FUNCTION_BLOCK E_F_TRIG
  (* Version 1.0, 2005-07-05, Goran Cengic, Chalmers *)
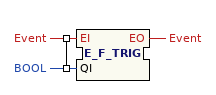
  EVENT_INPUT
    EI WITH QI;
  END_EVENT
  EVENT_OUTPUT
    EO;
  END_EVENT
  VAR_INPUT
    QI : BOOL;
  END_VAR
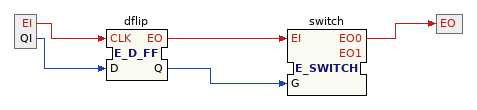
  FBS
    dflip : E_D_FF;
    switch : E_SWITCH;
  END_FBS
  EVENT_CONNECTIONS
    EI TO dflip.CLK;
    dflip.EO TO switch.EI;
    switch.EO0 TO EO;
  END_CONNECTIONS
  DATA_CONNECTIONS
    QI TO dflip.D;
    dflip.Q TO switch.G;
  END_CONNECTIONS
END_FUNCTION_BLOCK
